(* IEC 61131-3 sources: SmartHomeNew/snapshots/2026-05-12 (part 2) *)

(* ---- FB_Time_Service.st ---- *)
FUNCTION_BLOCK FB_Time_Service
VAR
    L_Real_Now : UDINT;
    L_Elapsed : UDINT;
    L_Scaled_Delta : UDINT;
END_VAR

// read real time
L_Real_Now := GVL_STATUS.G_System_Time_MS;

// wrap-safe delta (real time base)
IF L_Real_Now >= GVL_TIME_SERVICE.G_Last_Now_MS THEN
    L_Elapsed := L_Real_Now - GVL_TIME_SERVICE.G_Last_Now_MS;
    GVL_TIME_SERVICE.G_Wrap_Detected := FALSE;
ELSE
    L_Elapsed := (16#FFFFFFFF - GVL_TIME_SERVICE.G_Last_Now_MS) + L_Real_Now + 1;
    GVL_TIME_SERVICE.G_Wrap_Detected := TRUE;
END_IF;

GVL_TIME_SERVICE.G_Last_Now_MS := L_Real_Now;

// --- SIMULATION MODE ---
IF GVL_TIME_SERVICE.G_Sim_Enabled THEN

    IF NOT GVL_TIME_SERVICE.G_Sim_Frozen THEN
        L_Scaled_Delta := REAL_TO_UDINT(TO_REAL(L_Elapsed) * GVL_TIME_SERVICE.G_Sim_Time_Scale);

        GVL_TIME_SERVICE.G_Sim_Now_MS := GVL_TIME_SERVICE.G_Sim_Now_MS + L_Scaled_Delta;

        GVL_TIME_SERVICE.G_Sim_Time_Of_Day_MS := GVL_TIME_SERVICE.G_Sim_Time_Of_Day_MS + L_Scaled_Delta;

        IF GVL_TIME_SERVICE.G_Sim_Time_Of_Day_MS >= 86400000 THEN
            GVL_TIME_SERVICE.G_Sim_Time_Of_Day_MS := GVL_TIME_SERVICE.G_Sim_Time_Of_Day_MS MOD 86400000;
            GVL_TIME_SERVICE.G_Sim_Day_Of_Week := GVL_TIME_SERVICE.G_Sim_Day_Of_Week + 1;
            IF GVL_TIME_SERVICE.G_Sim_Day_Of_Week > 7 THEN
                GVL_TIME_SERVICE.G_Sim_Day_Of_Week := 1;
            END_IF;
        END_IF;
    END_IF;

    GVL_TIME_SERVICE.G_Now_MS := GVL_TIME_SERVICE.G_Sim_Now_MS;
    GVL_TIME_SERVICE.G_Time_Of_Day_MS := GVL_TIME_SERVICE.G_Sim_Time_Of_Day_MS;
    GVL_TIME_SERVICE.G_Day_Of_Week := GVL_TIME_SERVICE.G_Sim_Day_Of_Week;

ELSE
    GVL_TIME_SERVICE.G_Now_MS := L_Real_Now;
    GVL_TIME_SERVICE.G_Time_Of_Day_MS := GVL_STATUS.G_Time_Of_Day_MS;
    GVL_TIME_SERVICE.G_Day_Of_Week := TO_INT(GVL_STATUS.G_Current_Day);
END_IF;

// TOD unified
GVL_TIME_SERVICE.G_Current_TOD := UDINT_TO_TOD(GVL_TIME_SERVICE.G_Time_Of_Day_MS);

GVL_TIME_SERVICE.G_Delta_MS := L_Elapsed;

END_FUNCTION_BLOCK

(* ---- FB_Water_Output_Projection.st ---- *)
FUNCTION_BLOCK FB_Water_Output_Projection
VAR_INPUT
    VI_Zone_Enable : ARRAY[1..32] OF BOOL;
    VI_Valve_35_Close : BOOL;
    VI_Valve_36_Close : BOOL;
END_VAR
VAR
    L_i : INT;
END_VAR

FOR L_i := 1 TO 32 DO
    GVL_WATER_OUTPUT.DO_Water_Zone_Enable[L_i] := VI_Zone_Enable[L_i];
END_FOR;

GVL_WATER_OUTPUT.DO_Water_Valve_35_Close := VI_Valve_35_Close;
GVL_WATER_OUTPUT.DO_Water_Valve_36_Close := VI_Valve_36_Close;

END_FUNCTION_BLOCK
// >>> BULK_SYNC_ANCHOR: FB_Water_Output_Projection <<<

(* ---- PRG_Command_Verifier.st ---- *)
PROGRAM PRG_Command_Verifier
VAR
    L_i : INT;
    L_Mismatch_Count : INT := 0;
    L_Runtime_Error : BOOL := FALSE;
    L_Runtime_Error_Code : UDINT := 0;
    L_Runtime_Error_Text : STRING(160) := '';
    L_Now_MS : UDINT;
    L_Prev_Runtime_Error : BOOL;
    L_Any_Manifold_Pump_On : BOOL;
    fbLog : FB_LogEvent;
END_VAR

L_Now_MS := GVL_STATUS.G_System_Time_MS;

// ===============================
// 1. COMMAND MISMATCH CHECK
// ===============================
L_Mismatch_Count := 0;

IF GVL_COMMAND.G_Gas_Valve_Close <> GVL_COMMAND_SHADOW.G_Gas_Valve_Close THEN L_Mismatch_Count := L_Mismatch_Count + 1; END_IF;
IF GVL_COMMAND.G_Boiler_Stop <> GVL_COMMAND_SHADOW.G_Boiler_Stop THEN L_Mismatch_Count := L_Mismatch_Count + 1; END_IF;
IF GVL_COMMAND.G_Vent_Stop <> GVL_COMMAND_SHADOW.G_Vent_Stop THEN L_Mismatch_Count := L_Mismatch_Count + 1; END_IF;
IF GVL_COMMAND.G_Supply_100_Req <> GVL_COMMAND_SHADOW.G_Supply_100_Req THEN L_Mismatch_Count := L_Mismatch_Count + 1; END_IF;
IF GVL_COMMAND.G_Supply_80_Req <> GVL_COMMAND_SHADOW.G_Supply_80_Req THEN L_Mismatch_Count := L_Mismatch_Count + 1; END_IF;
IF GVL_COMMAND.G_Vent_PV3_Boost <> GVL_COMMAND_SHADOW.G_Vent_PV3_Boost THEN L_Mismatch_Count := L_Mismatch_Count + 1; END_IF;
IF GVL_COMMAND.G_Close_Valve_35 <> GVL_COMMAND_SHADOW.G_Close_Valve_35 THEN L_Mismatch_Count := L_Mismatch_Count + 1; END_IF;
IF GVL_COMMAND.G_Close_Valve_36 <> GVL_COMMAND_SHADOW.G_Close_Valve_36 THEN L_Mismatch_Count := L_Mismatch_Count + 1; END_IF;
IF GVL_COMMAND.G_Lock_1_Open <> GVL_COMMAND_SHADOW.G_Lock_1_Open THEN L_Mismatch_Count := L_Mismatch_Count + 1; END_IF;
IF GVL_COMMAND.G_Lock_1_Close <> GVL_COMMAND_SHADOW.G_Lock_1_Close THEN L_Mismatch_Count := L_Mismatch_Count + 1; END_IF;
IF GVL_COMMAND.G_Lock_2_Open <> GVL_COMMAND_SHADOW.G_Lock_2_Open THEN L_Mismatch_Count := L_Mismatch_Count + 1; END_IF;
IF GVL_COMMAND.G_Lock_2_Close <> GVL_COMMAND_SHADOW.G_Lock_2_Close THEN L_Mismatch_Count := L_Mismatch_Count + 1; END_IF;
IF GVL_COMMAND.G_Gate_Open <> GVL_COMMAND_SHADOW.G_Gate_Open THEN L_Mismatch_Count := L_Mismatch_Count + 1; END_IF;
IF GVL_COMMAND.G_Wicket_Open <> GVL_COMMAND_SHADOW.G_Wicket_Open THEN L_Mismatch_Count := L_Mismatch_Count + 1; END_IF;

GVL_COMMAND_VERIFY.Command_Mismatch_Count := L_Mismatch_Count;
GVL_COMMAND_VERIFY.Command_Match_OK := (L_Mismatch_Count = 0);
GVL_COMMAND_VERIFY.Command_Mismatch_Active := (L_Mismatch_Count > 0);

// ===============================
// 2. RUNTIME SANITY CHECKS
// ===============================
L_Runtime_Error := FALSE;
L_Runtime_Error_Code := 0;
L_Runtime_Error_Text := '';
L_Any_Manifold_Pump_On := FALSE;

// PLC inactive: fail-safe outputs should be off/safe except alarm/gas close outputs.
IF (NOT L_Runtime_Error) AND (NOT GVL_STATUS.G_Is_Active_PLC) THEN
    FOR L_i := 1 TO GVL_CONSTANTS.C_MAX_HEATING_CIRCUITS DO
        IF GVL_IO.DO_Zone_Valves[L_i] THEN
            L_Runtime_Error := TRUE;
            L_Runtime_Error_Code := 10;
            L_Runtime_Error_Text := 'PLC inactive zone valve on';
        END_IF;
    END_FOR;
END_IF;

IF (NOT L_Runtime_Error) AND (NOT GVL_STATUS.G_Is_Active_PLC) THEN
    FOR L_i := 1 TO GVL_CONSTANTS.C_MAX_MANIFOLDS DO
        IF GVL_IO.DO_Manifold_Pumps[L_i] THEN
            L_Runtime_Error := TRUE;
            L_Runtime_Error_Code := 11;
            L_Runtime_Error_Text := 'PLC inactive pump on';
        END_IF;
    END_FOR;
END_IF;

// GAS: gas valve must be physically commanded closed.
IF (NOT L_Runtime_Error) AND (GVL_SAFETY_SHUTDOWN.G_Safety_Mode = GAS) AND (NOT GVL_IO.DO_Gas_Valve_Close) THEN
    L_Runtime_Error := TRUE;
    L_Runtime_Error_Code := 1;
    L_Runtime_Error_Text := 'Gas valve not closed';
END_IF;

// GAS: ventilation must not be forced fully off by the IO layer.
IF (NOT L_Runtime_Error) AND (GVL_SAFETY_SHUTDOWN.G_Safety_Mode = GAS) THEN
    IF (GVL_IO.AO_Supply_Fans[1] = 0) AND (GVL_IO.AO_Exhaust_Fans[1] = 0) THEN
        L_Runtime_Error := TRUE;
        L_Runtime_Error_Code := 3;
        L_Runtime_Error_Text := 'Gas ventilation inactive';
    END_IF;
END_IF;

// FIRE: all exhaust fans should be commanded above zero in smoke exhaust mode.
IF (NOT L_Runtime_Error) AND (GVL_SAFETY_SHUTDOWN.G_Safety_Mode = FIRE) THEN
    FOR L_i := 1 TO GVL_CONSTANTS.C_MAX_EXHAUST_FANS DO
        IF GVL_IO.AO_Exhaust_Fans[L_i] = 0 THEN
            L_Runtime_Error := TRUE;
            L_Runtime_Error_Code := 2;
            L_Runtime_Error_Text := 'Smoke exhaust not active';
        END_IF;
    END_FOR;
END_IF;

// FIRE: supply fans should be off in smoke exhaust mode.
IF (NOT L_Runtime_Error) AND (GVL_SAFETY_SHUTDOWN.G_Safety_Mode = FIRE) THEN
    FOR L_i := 1 TO GVL_CONSTANTS.C_MAX_SUPPLY_FANS DO
        IF GVL_IO.AO_Supply_Fans[L_i] <> 0 THEN
            L_Runtime_Error := TRUE;
            L_Runtime_Error_Code := 4;
            L_Runtime_Error_Text := 'Supply fan active in fire';
        END_IF;
    END_FOR;
END_IF;

// WATER_LEAK: valve close commands must reach physical outputs.
IF (NOT L_Runtime_Error) AND (GVL_SAFETY_SHUTDOWN.G_Safety_Mode = WATER_LEAK) THEN
    IF GVL_COMMAND_SHADOW.G_Close_Valve_35 AND (NOT GVL_IO.DO_Water_Valve_35_Close) THEN
        L_Runtime_Error := TRUE;
        L_Runtime_Error_Code := 5;
        L_Runtime_Error_Text := 'Water valve 35 not closed';
    ELSIF GVL_COMMAND_SHADOW.G_Close_Valve_36 AND (NOT GVL_IO.DO_Water_Valve_36_Close) THEN
        L_Runtime_Error := TRUE;
        L_Runtime_Error_Code := 6;
        L_Runtime_Error_Text := 'Water valve 36 not closed';
    END_IF;
END_IF;

// FREEZE: when freeze-risk is active, heating circulation should not be fully dead.
IF (NOT L_Runtime_Error) AND GVL_STATE.G_Safety_Freeze_Risk THEN
    FOR L_i := 1 TO GVL_CONSTANTS.C_MAX_MANIFOLDS DO
        IF GVL_IO.DO_Manifold_Pumps[L_i] THEN
            L_Any_Manifold_Pump_On := TRUE;
        END_IF;
    END_FOR;

    IF (NOT L_Any_Manifold_Pump_On) AND (NOT GVL_IO.DO_Backup_Circulation_Pump) THEN
        L_Runtime_Error := TRUE;
        L_Runtime_Error_Code := 7;
        L_Runtime_Error_Text := 'Freeze circulation inactive';
    END_IF;
END_IF;

// GAS+FREEZE: electric backup may be used for anti-freeze, but DHW heating must remain off.
IF (NOT L_Runtime_Error) AND GVL_STATE.G_Safety_Freeze_Risk AND GVL_COMMAND_SHADOW.G_Heating_Gas_Safety_Stop THEN
    IF GVL_IO.DO_DHW_Heating_Pump THEN
        L_Runtime_Error := TRUE;
        L_Runtime_Error_Code := 8;
        L_Runtime_Error_Text := 'DHW heating active during gas freeze';
    END_IF;
END_IF;

// Apply result
IF L_Runtime_Error THEN
    GVL_COMMAND_VERIFY.Runtime_Sanity_OK := FALSE;
    GVL_COMMAND_VERIFY.Runtime_Last_Error_Code := L_Runtime_Error_Code;
    GVL_COMMAND_VERIFY.Runtime_Last_Error_Text := L_Runtime_Error_Text;
    GVL_COMMAND_VERIFY.Runtime_Last_Error_Time_MS := L_Now_MS;
    GVL_CONFIG_VALIDATION.G_Runtime_Sanity_OK := FALSE;
    GVL_CONFIG_VALIDATION.G_Runtime_Sanity_Error := TRUE;
    GVL_CONFIG_VALIDATION.G_Runtime_Last_Error_Code := L_Runtime_Error_Code;
    GVL_CONFIG_VALIDATION.G_Runtime_Last_Error_Text := L_Runtime_Error_Text;
    GVL_CONFIG_VALIDATION.G_Runtime_Last_Error_MS := L_Now_MS;

    IF NOT L_Prev_Runtime_Error THEN
        GVL_COMMAND_VERIFY.Runtime_Sanity_Error_Count := GVL_COMMAND_VERIFY.Runtime_Sanity_Error_Count + 1;
        fbLog(
            VI_Event_Type := 1001,
            VI_Timestamp := L_Now_MS,
            VI_Param1 := L_Runtime_Error_Code,
            VI_Param2 := GVL_COMMAND_VERIFY.Runtime_Sanity_Error_Count
        );
    END_IF;
ELSE
    GVL_COMMAND_VERIFY.Runtime_Sanity_OK := TRUE;
    GVL_CONFIG_VALIDATION.G_Runtime_Sanity_OK := TRUE;
    GVL_CONFIG_VALIDATION.G_Runtime_Sanity_Error := FALSE;
END_IF;

L_Prev_Runtime_Error := L_Runtime_Error;

END_PROGRAM

(* ---- PRG_Config_Versioning.st ---- *)
PROGRAM PRG_Config_Versioning
VAR
    L_i : INT;
    L_Config_Error : BOOL;
END_VAR

// Detect config error from validation layer
L_Config_Error := GVL_STATUS.G_Diagnostics.Sensor_Fault OR GVL_STATUS.G_Diagnostics.Subsystem_Degraded;

// --- Save snapshot when system is healthy ---
IF NOT L_Config_Error THEN
    FOR L_i := 1 TO GVL_CONSTANTS.C_MAX_HEATING_CIRCUITS DO
        GVL_CONFIG_BACKUP.G_Backup_FloorHeating_Configs[L_i] := GVL_CONFIG.G_HMI_FloorHeating_Configs[L_i];
    END_FOR;

    GVL_CONFIG_BACKUP.G_Backup_Max_Active_Manifolds := GVL_CONFIG.G_Max_Active_Manifolds;
    GVL_CONFIG_BACKUP.G_Backup_Max_Thermal_Budget := GVL_CONFIG.G_Max_Thermal_Budget;

    GVL_CONFIG_BACKUP.G_Backup_Valid := TRUE;
END_IF;

// --- Rollback if config invalid ---
IF L_Config_Error THEN

    // Freeze system via command layer
    GVL_COMMAND_SHADOW.G_Heating_Block := TRUE;
    GVL_COMMAND_SHADOW.G_Boiler_Stop := TRUE;

    // Restore snapshot only if valid
    IF GVL_CONFIG_BACKUP.G_Backup_Valid THEN
        FOR L_i := 1 TO GVL_CONSTANTS.C_MAX_HEATING_CIRCUITS DO
            GVL_CONFIG.G_HMI_FloorHeating_Configs[L_i] := GVL_CONFIG_BACKUP.G_Backup_FloorHeating_Configs[L_i];
        END_FOR;

        GVL_CONFIG.G_Max_Active_Manifolds := GVL_CONFIG_BACKUP.G_Backup_Max_Active_Manifolds;
        GVL_CONFIG.G_Max_Thermal_Budget := GVL_CONFIG_BACKUP.G_Backup_Max_Thermal_Budget;

        GVL_STATUS.G_System_Mode_Text := 'CONFIG ROLLBACK';
    ELSE
        GVL_STATUS.G_System_Mode_Text := 'CONFIG INVALID - NO BACKUP';
    END_IF;
END_IF;

END_PROGRAM
// >>> BULK_SYNC_ANCHOR: PRG_Config_Versioning <<<

(* ---- PRG_Explainability.st ---- *)
PROGRAM PRG_Explainability
VAR
    L_Mode : E_Safety_Mode;
    L_Recovery : E_Recovery_Phase;
    L_Command : STRING(120);
    L_Heating : STRING(255);
END_VAR

L_Mode := GVL_SAFETY_SHUTDOWN.G_Safety_Mode;
L_Recovery := GVL_SAFETY_RECOVERY.G_Recovery_Phase;

GVL_EXPLAINABILITY.G_Last_Safety_Mode := L_Mode;
GVL_EXPLAINABILITY.G_Last_Recovery_Phase := L_Recovery;
GVL_EXPLAINABILITY.G_Last_Update_MS := GVL_TIME_SERVICE.G_Now_MS;

// SAFETY LEVEL
CASE L_Mode OF
    FIRE: GVL_EXPLAINABILITY.G_Reason_Chain_Safety := 'FIRE';
    GAS: GVL_EXPLAINABILITY.G_Reason_Chain_Safety := 'GAS';
    WATER_LEAK: GVL_EXPLAINABILITY.G_Reason_Chain_Safety := 'WATER';
    GLOBAL_STOP: GVL_EXPLAINABILITY.G_Reason_Chain_Safety := 'GLOBAL_STOP';
    ELSE
        IF GVL_SAFETY_RECOVERY.G_Recovery_Active THEN
            GVL_EXPLAINABILITY.G_Reason_Chain_Safety := 'RECOVERY';
        ELSE
            GVL_EXPLAINABILITY.G_Reason_Chain_Safety := 'NORMAL';
        END_IF;
END_CASE;

// BEHAVIOR LEVEL
GVL_EXPLAINABILITY.G_Reason_Chain_Behavior := GVL_INTENT_BEHAVIOR.I_Reason_Text;

// COMMAND LEVEL
IF GVL_COMMAND_SHADOW.G_Heating_Block THEN
    L_Command := 'Heating Blocked';
ELSIF GVL_COMMAND_SHADOW.G_Vent_Stop THEN
    L_Command := 'Vent Stopped';
ELSIF GVL_COMMAND_SHADOW.G_Water_Block THEN
    L_Command := 'Water Blocked';
ELSE
    L_Command := 'Command OK';
END_IF;
GVL_EXPLAINABILITY.G_Reason_Chain_Command := L_Command;

// HEATING DOMAIN EXPLAINABILITY
IF GVL_STATE.G_Heating_RootCause <> E_Heating_RootCause.RC_NONE THEN
    L_Heating := GVL_STATE.G_Heating_Confidence_Reason_Text;
ELSIF GVL_STATE.G_Heating_Cascade_Degraded THEN
    L_Heating := 'Heating cascade degraded';
ELSE
    L_Heating := 'Heating OK';
END_IF;
GVL_EXPLAINABILITY.G_Heating_Why_Blocked := L_Heating;

// OUTPUT LEVEL
GVL_EXPLAINABILITY.G_Reason_Chain_Output := 'Outputs Applied';

// FULL CHAIN
GVL_EXPLAINABILITY.G_Reason_Chain_Full := CONCAT(
    CONCAT(
        CONCAT(
            GVL_EXPLAINABILITY.G_Reason_Chain_Safety,
            ' -> '
        ),
        CONCAT(
            GVL_EXPLAINABILITY.G_Reason_Chain_Behavior,
            ' -> '
        )
    ),
    CONCAT(
        CONCAT(
            GVL_EXPLAINABILITY.G_Reason_Chain_Command,
            ' -> '
        ),
        CONCAT(
            L_Heating,
            ' -> Outputs Applied'
        )
    )
);

// KEEP OLD FIELDS
GVL_EXPLAINABILITY.G_Behavior_Why_Active := GVL_INTENT_BEHAVIOR.I_Reason_Text;

END_PROGRAM

(* ---- PRG_Heating.st ---- *)
PROGRAM PRG_Heating
VAR
    fbHeatingManager : FB_Heating_System_Manager;
    fbDHWManager : FB_DHW_Manager;
    fbOutputProjection : FB_Heating_Output_Projection;
    fbRootCauseDiagnostics : FB_Heating_RootCause_Diagnostics;
    fbHeatingDiagnostics : FB_Heating_Diagnostics;
    fbRuntimeObserver : FB_Heating_Runtime_Observer;
    fbRuntimeObserverAuthorization : FB_Heating_Runtime_Observer_Authorization;

    L_Runtime_Context : ST_Heating_Runtime_Context;

    L_Runtime_Observer_Enable_Last : BOOL := FALSE;
    L_Runtime_Observer_Activation_Stabilized : BOOL := FALSE;

    L_i : INT;
    L_Current_Hour : UINT;
    L_Boiler_Modulation_REAL : ARRAY[1..GVL_CONSTANTS.C_MAX_BOILERS] OF REAL;

    L_Heating_Emergency_Stop : BOOL;
    L_Heating_Gas_Safety_Stop : BOOL;

    L_Zone_Valves : ARRAY[1..GVL_CONSTANTS.C_MAX_HEATING_CIRCUITS] OF BOOL;
    L_Manifold_Pumps : ARRAY[1..GVL_CONSTANTS.C_MAX_MANIFOLDS] OF BOOL;
    L_Manifold_Valves : ARRAY[1..GVL_CONSTANTS.C_MAX_MANIFOLDS] OF REAL;
    L_Boiler_OT_Enable : ARRAY[1..GVL_CONSTANTS.C_MAX_BOILERS] OF BOOL;
    L_Boiler_OT_Setpoint : ARRAY[1..GVL_CONSTANTS.C_MAX_BOILERS] OF REAL;
    L_Backup_Circulation_Pump : BOOL;
    L_Electric_Heater_Enable : BOOL;
    L_Freeze_Risk_Status : BOOL;
    L_Manifold_Status : ARRAY[1..GVL_CONSTANTS.C_MAX_MANIFOLDS] OF ST_Manifold_Status;
    L_Boiler_Status : ARRAY[1..GVL_CONSTANTS.C_MAX_BOILERS] OF ST_Boiler_Status;
    L_DHW_Heating_Pump : BOOL;
    L_DHW_Circ_Pump : BOOL;
    L_DHW_Status : ST_DHW_Status;
END_VAR

FOR L_i := 1 TO GVL_CONSTANTS.C_MAX_BOILERS DO
    L_Boiler_Modulation_REAL[L_i] := TO_REAL(GVL_IO.AI_Boiler_Modulation[L_i]);
END_FOR;

L_Current_Hour := TO_UINT(GVL_TIME_SERVICE.G_Time_Of_Day_MS / 3600000);

L_Heating_Emergency_Stop := GVL_COMMAND_SHADOW.G_Heating_Emergency_Stop;
L_Heating_Gas_Safety_Stop := GVL_COMMAND_SHADOW.G_Heating_Gas_Safety_Stop OR GVL_STATE.G_Safety_Gas_Latched;

L_Runtime_Context.Runtime_Enabled := TRUE;
L_Runtime_Context.Runtime_Ready := TRUE;
L_Runtime_Context.Runtime_Fault := FALSE;
L_Runtime_Context.Current_Phase := E_Heating_Runtime_Phase.HRP_IDLE;

L_Runtime_Context.Allow_DHW_Phase := TRUE;
L_Runtime_Context.Allow_Heating_Phase := TRUE;
L_Runtime_Context.Allow_Service_Gating_Phase := TRUE;
L_Runtime_Context.Allow_State_Publication_Phase := TRUE;
L_Runtime_Context.Allow_Diagnostics_Phase := TRUE;
L_Runtime_Context.Allow_Output_Projection_Phase := TRUE;

L_Runtime_Context.DHW_Executed := FALSE;
L_Runtime_Context.Heating_Executed := FALSE;
L_Runtime_Context.Service_Gating_Executed := FALSE;
L_Runtime_Context.State_Publication_Executed := FALSE;
L_Runtime_Context.Diagnostics_Executed := FALSE;
L_Runtime_Context.Output_Projection_Executed := FALSE;

L_Runtime_Context.DHW_Before_Heating_Valid := TRUE;
L_Runtime_Context.State_Publication_Before_Diagnostics_Valid := TRUE;
L_Runtime_Context.Output_Projection_Last_Valid := TRUE;

L_Runtime_Context.Diagnostics_Isolation_Valid := TRUE;
L_Runtime_Context.Explainability_Isolation_Valid := TRUE;
L_Runtime_Context.Safety_Isolation_Valid := TRUE;
L_Runtime_Context.OpenTherm_Ownership_Valid := TRUE;
L_Runtime_Context.Cascade_Ownership_Valid := TRUE;

L_Runtime_Context.Runtime_Status_Code := 1;
L_Runtime_Context.Runtime_Status_Text := 'Heating runtime nominal';

// ======================================================
// GOVERNED OBSERVER AUTHORIZATION EVALUATION
// ======================================================
GVL_Heating_Runtime_Observer.G_Runtime_Observer_Lifecycle_State :=
    E_Runtime_Observer_Lifecycle_State.ROS_AUTHORIZATION_PENDING;
GVL_Heating_Runtime_Observation.G_Runtime_Observer_Lifecycle_State :=
    E_Runtime_Observer_Lifecycle_State.ROS_AUTHORIZATION_PENDING;
GVL_Heating_Runtime_Observation.G_Runtime_Observer_Lifecycle_Code := 10;
GVL_Heating_Runtime_Observation.G_Runtime_Observer_Lifecycle_Text :=
    'Heating runtime observer authorization pending';
GVL_Heating_Runtime_Observation.G_Runtime_Observer_Commissioning_Active :=
    GVL_Heating_Runtime_Observer.G_Runtime_Observer_Enable_Request;

fbRuntimeObserverAuthorization(
    VI_Enable_Request := GVL_Heating_Runtime_Observer.G_Runtime_Observer_Enable_Request,
    VI_Bootstrap_Mode := GVL_Heating_Runtime_Observer.G_Runtime_Observer_Bootstrap_Mode,
    VI_Passive_Mode := GVL_Heating_Runtime_Observer.G_Runtime_Observer_Passive_Mode,
    VI_ReadOnly_Mode := GVL_Heating_Runtime_Observer.G_Runtime_Observer_ReadOnly_Mode,
    VI_Governance_Locked := GVL_Heating_Runtime_Observer.G_Runtime_Observer_Governance_Locked,
    VI_Runtime_Authority_Disabled := GVL_Heating_Runtime_Observer.G_Runtime_Observer_Runtime_Authority_Disabled,
    VI_Writable_Exports_Disabled := GVL_Heating_Runtime_Observer.G_Runtime_Observer_Writable_Exports_Disabled
);

GVL_Heating_Runtime_Observer.G_Runtime_Observer_Enable_Authorized :=
    fbRuntimeObserverAuthorization.VO_Enable_Authorized;

GVL_Heating_Runtime_Observer.G_Runtime_Observer_Enable_Effective :=
    fbRuntimeObserverAuthorization.VO_Enable_Effective;

GVL_Heating_Runtime_Observer.G_Runtime_Observer_Authorization_Valid :=
    fbRuntimeObserverAuthorization.VO_Authorization_Valid;

GVL_Heating_Runtime_Observer.G_Runtime_Observer_Authorization_Status_Code :=
    fbRuntimeObserverAuthorization.VO_Status_Code;

GVL_Heating_Runtime_Observer.G_Runtime_Observer_Authorization_Status_Text :=
    fbRuntimeObserverAuthorization.VO_Status_Text;

IF NOT GVL_Heating_Runtime_Observer.G_Runtime_Observer_Enable_Request THEN
    GVL_Heating_Runtime_Observer.G_Runtime_Observer_Lifecycle_State :=
        E_Runtime_Observer_Lifecycle_State.ROS_INACTIVE;
    GVL_Heating_Runtime_Observation.G_Runtime_Observer_Lifecycle_State :=
        E_Runtime_Observer_Lifecycle_State.ROS_INACTIVE;
    GVL_Heating_Runtime_Observation.G_Runtime_Observer_Lifecycle_Code := 0;
    GVL_Heating_Runtime_Observation.G_Runtime_Observer_Lifecycle_Text :=
        'Heating runtime observer inactive';
    GVL_Heating_Runtime_Observation.G_Runtime_Observer_Commissioning_Active := FALSE;
ELSIF NOT GVL_Heating_Runtime_Observer.G_Runtime_Observer_Enable_Effective THEN
    GVL_Heating_Runtime_Observer.G_Runtime_Observer_Lifecycle_State :=
        E_Runtime_Observer_Lifecycle_State.ROS_AUTHORIZATION_DENIED;
    GVL_Heating_Runtime_Observation.G_Runtime_Observer_Lifecycle_State :=
        E_Runtime_Observer_Lifecycle_State.ROS_AUTHORIZATION_DENIED;
    GVL_Heating_Runtime_Observation.G_Runtime_Observer_Lifecycle_Code := 20;
    GVL_Heating_Runtime_Observation.G_Runtime_Observer_Lifecycle_Text :=
        'Heating runtime observer authorization denied';
END_IF;

L_Runtime_Context.Current_Phase := E_Heating_Runtime_Phase.HRP_DHW;

fbDHWManager(
    VI_System_Time_MS := GVL_STATUS.G_System_Time_MS,
    VI_Current_TOD := GVL_STATUS.G_Current_TOD,
    VI_IsActivePLC := GVL_STATUS.G_Is_Active_PLC,
    VI_Temp := GVL_STATE.G_DHW_Temp,
    VI_Pressure := GVL_STATE.G_DHW_Pressure,
    VI_Config := GVL_CONFIG.G_DHW_Config,
    VI_Current_Day_Of_Week := GVL_STATUS.G_Current_Day,
    VI_IO_Modules_Online := GVL_STATUS.G_IO_Modules_Online,
    VI_Reset_Errors := GVL_INTENT_USER.I_Reset_Errors,
    VI_Emergency_Stop := L_Heating_Emergency_Stop,
    VI_System_Mode := GVL_STATE.G_System_Mode,
    VO_Status => L_DHW_Status,
    VO_Heating_Pump => L_DHW_Heating_Pump,
    VO_Circ_Pump => L_DHW_Circ_Pump
);

L_Runtime_Context.DHW_Executed := TRUE;

IF L_Heating_Gas_Safety_Stop THEN
    L_DHW_Heating_Pump := FALSE;
    L_DHW_Status.Heating_Pump_On := FALSE;
END_IF;

L_Runtime_Context.Current_Phase := E_Heating_Runtime_Phase.HRP_HEATING;

fbHeatingManager(
    VI_System_Mode := GVL_STATE.G_System_Mode,
    VI_System_Time_MS := GVL_STATUS.G_System_Time_MS,
    VI_IsActivePLC := GVL_STATUS.G_Is_Active_PLC,
    VI_Outdoor_Temp := GVL_STATE.G_Outdoor_Temp,
    VI_Config := GVL_CONFIG.G_Heating_Config,
    VI_Tariff := GVL_CONFIG.G_HMI_Tariff_Settings,
    VI_Current_Hour := L_Current_Hour,
    VI_DHW_Heating_Demand := L_DHW_Heating_Pump,
    VI_DHW_Target_Temp := GVL_CONFIG.G_DHW_Config.Target_Temp,
    VI_Emergency_Stop := L_Heating_Emergency_Stop,
    VI_Gas_Safety_Stop := L_Heating_Gas_Safety_Stop,
    VI_Boiler_Error_Status := GVL_STATE.G_Boiler_Error,
    VI_Boiler_OT_Online := GVL_STATE.G_Boiler_OT_Online,
    VI_Boiler_Modulation := L_Boiler_Modulation_REAL,
    VI_Floor_Temps := GVL_STATE.G_Floor_Temps,
    VI_Room_Temps := GVL_STATE.G_Room_Temps,
    VI_Manifold_Pressures := GVL_STATE.G_Manifold_Pressures,
    VI_Manifold_Currents := GVL_STATE.G_Manifold_Currents,
    VI_Manifold_Temps_Supply := GVL_STATE.G_Manifold_T_Supply,
    VI_Manifold_Temps_Return := GVL_STATE.G_Manifold_T_Return,
    VI_Boiler_Flame_Status := GVL_STATE.G_Boiler_Flame,
    VI_Zone_Configs := GVL_CONFIG.G_HMI_FloorHeating_Configs,
    VI_Rule_Actions := GVL_STATE.G_Rule_Actions,
    VI_IO_Modules_Online := GVL_STATUS.G_IO_Modules_Online,
    VI_Manifold_End_Switches := GVL_STATE.G_Manifold_End_Switches,
    VI_Valve_Test_Config := GVL_CONFIG.G_Valve_Test_Config,
    VO_Manifold_Valves => L_Manifold_Valves,
    VO_Manifold_Pumps => L_Manifold_Pumps,
    VO_Zone_Valves => L_Zone_Valves,
    VO_Boiler_OT_Enable => L_Boiler_OT_Enable,
    VO_Boiler_OT_Setpoint => L_Boiler_OT_Setpoint,
    VO_Backup_Circulation_Pump => L_Backup_Circulation_Pump,
    VO_Electric_Heater_Enable => L_Electric_Heater_Enable,
    VO_Freeze_Risk_Status => L_Freeze_Risk_Status,
    VO_Status => L_Manifold_Status,
    VO_Boiler_Status => L_Boiler_Status
);

L_Runtime_Context.Heating_Executed := TRUE;

L_Runtime_Context.Current_Phase := E_Heating_Runtime_Phase.HRP_SERVICE_GATING;

GVL_STATUS.G_Diagnostics.Backup_Pump_Out_Of_Service := NOT GVL_CONFIG.G_Backup_Circulation_Pump_In_Service;
GVL_STATUS.G_Diagnostics.Electric_Heater_Out_Of_Service := NOT GVL_CONFIG.G_Electric_Heater_In_Service;

IF NOT GVL_CONFIG.G_Backup_Circulation_Pump_In_Service THEN
    L_Backup_Circulation_Pump := FALSE;
END_IF;

IF NOT GVL_CONFIG.G_Electric_Heater_In_Service THEN
    L_Electric_Heater_Enable := FALSE;
END_IF;

FOR L_i := 1 TO GVL_CONSTANTS.C_MAX_MANIFOLDS DO
    GVL_STATUS.G_Diagnostics.Manifold_Pump_Out_Of_Service[L_i] := NOT GVL_CONFIG.G_Manifold_Pump_In_Service[L_i];
    IF NOT GVL_CONFIG.G_Manifold_Pump_In_Service[L_i] THEN
        L_Manifold_Pumps[L_i] := FALSE;
    END_IF;
END_FOR;

GVL_STATUS.G_Diagnostics.DHW_Heating_Pump_Out_Of_Service := NOT GVL_CONFIG.G_DHW_Heating_Pump_In_Service;
IF NOT GVL_CONFIG.G_DHW_Heating_Pump_In_Service THEN
    L_DHW_Heating_Pump := FALSE;
    L_DHW_Status.Heating_Pump_On := FALSE;
END_IF;

GVL_STATUS.G_Diagnostics.DHW_Circ_Pump_Out_Of_Service := NOT GVL_CONFIG.G_DHW_Circ_Pump_In_Service;
IF NOT GVL_CONFIG.G_DHW_Circ_Pump_In_Service THEN
    L_DHW_Circ_Pump := FALSE;
    L_DHW_Status.Circ_Pump_On := FALSE;
END_IF;

GVL_STATE.G_Freeze_Hardware_Degraded := GVL_STATUS.G_Diagnostics.Backup_Pump_Fault OR GVL_STATUS.G_Diagnostics.Electric_Heater_Fault;
GVL_STATE.G_Freeze_Hardware_Failed := GVL_STATUS.G_Diagnostics.Backup_Pump_Fault AND GVL_STATUS.G_Diagnostics.Electric_Heater_Fault;

IF GVL_STATE.G_Freeze_Hardware_Failed THEN
    L_Backup_Circulation_Pump := FALSE;
    L_Electric_Heater_Enable := FALSE;
    L_Freeze_Risk_Status := TRUE;
END_IF;

L_Runtime_Context.Service_Gating_Executed := TRUE;

L_Runtime_Context.Current_Phase := E_Heating_Runtime_Phase.HRP_STATE_PUBLICATION;

FOR L_i := 1 TO GVL_CONSTANTS.C_MAX_HEATING_CIRCUITS DO
    GVL_STATE.G_Zone_Valves[L_i] := L_Zone_Valves[L_i];
END_FOR;

FOR L_i := 1 TO GVL_CONSTANTS.C_MAX_MANIFOLDS DO
    GVL_STATE.G_Manifold_Pumps[L_i] := L_Manifold_Pumps[L_i];
    GVL_STATE.G_Manifold_Valves[L_i] := L_Manifold_Valves[L_i];
    GVL_STATUS.G_Manifold_Status[L_i] := L_Manifold_Status[L_i];
END_FOR;

FOR L_i := 1 TO GVL_CONSTANTS.C_MAX_BOILERS DO
    GVL_STATE.G_Boiler_OT_Enable[L_i] := L_Boiler_OT_Enable[L_i];
    GVL_STATE.G_Boiler_OT_Setpoint[L_i] := L_Boiler_OT_Setpoint[L_i];
    GVL_STATUS.G_Boiler_Status[L_i] := L_Boiler_Status[L_i];
END_FOR;

GVL_STATE.G_Backup_Circulation_Pump := L_Backup_Circulation_Pump;
GVL_STATE.G_Electric_Heater_Enable := L_Electric_Heater_Enable;
GVL_STATE.G_Safety_Freeze_Risk := L_Freeze_Risk_Status;
GVL_STATE.G_DHW_Heating_Pump := L_DHW_Heating_Pump;
GVL_STATE.G_DHW_Circ_Pump := L_DHW_Circ_Pump;
GVL_STATUS.G_DHW_Status := L_DHW_Status;

L_Runtime_Context.State_Publication_Executed := TRUE;

L_Runtime_Context.Current_Phase := E_Heating_Runtime_Phase.HRP_DIAGNOSTICS;

fbRootCauseDiagnostics(
    VI_Enable := TRUE
);

fbHeatingDiagnostics(
    VI_System_Time_MS := GVL_STATUS.G_System_Time_MS
);

L_Runtime_Context.Diagnostics_Executed := TRUE;

// ======================================================
// GOVERNED FINALIZED-STATE RUNTIME OBSERVER
// ======================================================
IF GVL_Heating_Runtime_Observer.G_Runtime_Observer_Enable_Effective THEN

    GVL_Heating_Runtime_Observer.G_Runtime_Observer_Rollback_Validated := FALSE;

    IF NOT L_Runtime_Observer_Enable_Last THEN
        L_Runtime_Observer_Activation_Stabilized := FALSE;

        GVL_Heating_Runtime_Observer.G_Runtime_Observer_Lifecycle_State :=
            E_Runtime_Observer_Lifecycle_State.ROS_STABILIZATION;
        GVL_Heating_Runtime_Observation.G_Runtime_Observer_Lifecycle_State :=
            E_Runtime_Observer_Lifecycle_State.ROS_STABILIZATION;
        GVL_Heating_Runtime_Observation.G_Runtime_Observer_Lifecycle_Code := 30;
        GVL_Heating_Runtime_Observation.G_Runtime_Observer_Lifecycle_Text :=
            'Heating runtime observer stabilization active';

        GVL_Heating_Runtime_Observation.G_Runtime_Observer_Commissioning_Required := TRUE;
        GVL_Heating_Runtime_Observation.G_Runtime_Observer_Commissioning_Active := TRUE;
        GVL_Heating_Runtime_Observation.G_Runtime_Observer_Commissioning_Complete := FALSE;

        GVL_Heating_Runtime_Observation.G_Runtime_Observation_Publication_Valid := FALSE;
        GVL_Heating_Runtime_Observation.G_Runtime_Observation_Stabilization_Complete := FALSE;
        GVL_Heating_Runtime_Observation.G_Runtime_Observation_Operational := FALSE;

        GVL_Heating_Runtime_Observation.G_Runtime_Observation_Valid := FALSE;
        GVL_Heating_Runtime_Observation.G_Runtime_Observer_Ready := FALSE;
        GVL_Heating_Runtime_Observation.G_Runtime_Observer_Fault := FALSE;
        GVL_Heating_Runtime_Observation.G_Runtime_Observation_Status_Code := 100;
        GVL_Heating_Runtime_Observation.G_Runtime_Observation_Status_Text :=
            'Heating runtime observer stabilization cycle active';
    END_IF;

    fbRuntimeObserver(
        VI_Enable := TRUE,
        VI_Runtime_Context := L_Runtime_Context,
        VI_Diagnostics_Valid := TRUE
    );

    GVL_Heating_Runtime_Observation.G_Runtime_Observation :=
        fbRuntimeObserver.VO_Observation;

    IF L_Runtime_Observer_Activation_Stabilized THEN
        GVL_Heating_Runtime_Observer.G_Runtime_Observer_Lifecycle_State :=
            E_Runtime_Observer_Lifecycle_State.ROS_OPERATIONAL;
        GVL_Heating_Runtime_Observation.G_Runtime_Observer_Lifecycle_State :=
            E_Runtime_Observer_Lifecycle_State.ROS_OPERATIONAL;
        GVL_Heating_Runtime_Observation.G_Runtime_Observer_Lifecycle_Code := 40;
        GVL_Heating_Runtime_Observation.G_Runtime_Observer_Lifecycle_Text :=
            'Heating runtime observer operational';

        GVL_Heating_Runtime_Observation.G_Runtime_Observer_Commissioning_Required := FALSE;
        GVL_Heating_Runtime_Observation.G_Runtime_Observer_Commissioning_Active := FALSE;
        GVL_Heating_Runtime_Observation.G_Runtime_Observer_Commissioning_Complete := TRUE;

        GVL_Heating_Runtime_Observation.G_Runtime_Observation_Publication_Valid := TRUE;
        GVL_Heating_Runtime_Observation.G_Runtime_Observation_Stabilization_Complete := TRUE;
        GVL_Heating_Runtime_Observation.G_Runtime_Observation_Operational := TRUE;

        GVL_Heating_Runtime_Observation.G_Runtime_Observation_Valid := TRUE;
        GVL_Heating_Runtime_Observation.G_Runtime_Observer_Ready :=
            fbRuntimeObserver.VO_Observer_Ready;
        GVL_Heating_Runtime_Observation.G_Runtime_Observer_Fault :=
            fbRuntimeObserver.VO_Observer_Fault;
        GVL_Heating_Runtime_Observation.G_Runtime_Observation_Status_Code :=
            fbRuntimeObserver.VO_Status_Code;
        GVL_Heating_Runtime_Observation.G_Runtime_Observation_Status_Text :=
            fbRuntimeObserver.VO_Status_Text;

        GVL_Heating_Runtime_Observer.G_Runtime_Observer_Activation_Validated := TRUE;
        GVL_Heating_Runtime_Observer.G_Runtime_Observer_Sequencing_Validated := TRUE;
        GVL_Heating_Runtime_Observer.G_Runtime_Observer_Publication_Validated := TRUE;
    ELSE
        L_Runtime_Observer_Activation_Stabilized := TRUE;
    END_IF;

ELSE
    L_Runtime_Observer_Activation_Stabilized := FALSE;

    IF L_Runtime_Observer_Enable_Last THEN
        GVL_Heating_Runtime_Observer.G_Runtime_Observer_Lifecycle_State :=
            E_Runtime_Observer_Lifecycle_State.ROS_ROLLBACK;
        GVL_Heating_Runtime_Observation.G_Runtime_Observer_Lifecycle_State :=
            E_Runtime_Observer_Lifecycle_State.ROS_ROLLBACK;
        GVL_Heating_Runtime_Observation.G_Runtime_Observer_Lifecycle_Code := 50;
        GVL_Heating_Runtime_Observation.G_Runtime_Observer_Lifecycle_Text :=
            'Heating runtime observer rollback cleanup completed';
    ELSIF GVL_Heating_Runtime_Observer.G_Runtime_Observer_Enable_Request THEN
        GVL_Heating_Runtime_Observer.G_Runtime_Observer_Lifecycle_State :=
            E_Runtime_Observer_Lifecycle_State.ROS_AUTHORIZATION_DENIED;
        GVL_Heating_Runtime_Observation.G_Runtime_Observer_Lifecycle_State :=
            E_Runtime_Observer_Lifecycle_State.ROS_AUTHORIZATION_DENIED;
        GVL_Heating_Runtime_Observation.G_Runtime_Observer_Lifecycle_Code := 20;
        GVL_Heating_Runtime_Observation.G_Runtime_Observer_Lifecycle_Text :=
            'Heating runtime observer authorization denied';
    ELSE
        GVL_Heating_Runtime_Observer.G_Runtime_Observer_Lifecycle_State :=
            E_Runtime_Observer_Lifecycle_State.ROS_INACTIVE;
        GVL_Heating_Runtime_Observation.G_Runtime_Observer_Lifecycle_State :=
            E_Runtime_Observer_Lifecycle_State.ROS_INACTIVE;
        GVL_Heating_Runtime_Observation.G_Runtime_Observer_Lifecycle_Code := 0;
        GVL_Heating_Runtime_Observation.G_Runtime_Observer_Lifecycle_Text :=
            'Heating runtime observer inactive';
    END_IF;

    GVL_Heating_Runtime_Observation.G_Runtime_Observer_Commissioning_Required := TRUE;
    GVL_Heating_Runtime_Observation.G_Runtime_Observer_Commissioning_Active := FALSE;
    GVL_Heating_Runtime_Observation.G_Runtime_Observer_Commissioning_Complete := FALSE;

    GVL_Heating_Runtime_Observation.G_Runtime_Observation.Runtime_Active := FALSE;
    GVL_Heating_Runtime_Observation.G_Runtime_Observation.Runtime_Ready := FALSE;
    GVL_Heating_Runtime_Observation.G_Runtime_Observation.Runtime_Fault := FALSE;
    GVL_Heating_Runtime_Observation.G_Runtime_Observation.Current_Phase := E_Heating_Runtime_Phase.HRP_DISABLED;

    GVL_Heating_Runtime_Observation.G_Runtime_Observation.DHW_Demand_Active := FALSE;
    GVL_Heating_Runtime_Observation.G_Runtime_Observation.DHW_Heating_Active := FALSE;
    GVL_Heating_Runtime_Observation.G_Runtime_Observation.DHW_Circulation_Active := FALSE;

    GVL_Heating_Runtime_Observation.G_Runtime_Observation.Heating_Demand_Active := FALSE;
    GVL_Heating_Runtime_Observation.G_Runtime_Observation.Heating_Runtime_Active := FALSE;
    GVL_Heating_Runtime_Observation.G_Runtime_Observation.Heating_Output_Active := FALSE;

    GVL_Heating_Runtime_Observation.G_Runtime_Observation.Cascade_Available := FALSE;
    GVL_Heating_Runtime_Observation.G_Runtime_Observation.Cascade_Degraded := FALSE;
    GVL_Heating_Runtime_Observation.G_Runtime_Observation.Cascade_Active_Boilers := 0;
    GVL_Heating_Runtime_Observation.G_Runtime_Observation.Cascade_Available_Boilers := 0;

    GVL_Heating_Runtime_Observation.G_Runtime_Observation.OpenTherm_Online := FALSE;
    GVL_Heating_Runtime_Observation.G_Runtime_Observation.OpenTherm_Command_Valid := FALSE;
    GVL_Heating_Runtime_Observation.G_Runtime_Observation.OpenTherm_Transport_Degraded := FALSE;

    GVL_Heating_Runtime_Observation.G_Runtime_Observation.Diagnostics_Active := FALSE;
    GVL_Heating_Runtime_Observation.G_Runtime_Observation.Explainability_Active := FALSE;

    GVL_Heating_Runtime_Observation.G_Runtime_Observation.DHW_Before_Heating_Observed := FALSE;
    GVL_Heating_Runtime_Observation.G_Runtime_Observation.Diagnostics_After_Publication_Observed := FALSE;
    GVL_Heating_Runtime_Observation.G_Runtime_Observation.Output_Projection_Last_Observed := FALSE;

    GVL_Heating_Runtime_Observation.G_Runtime_Observation.Runtime_Ownership_Valid := FALSE;
    GVL_Heating_Runtime_Observation.G_Runtime_Observation.Diagnostics_Ownership_Valid := FALSE;
    GVL_Heating_Runtime_Observation.G_Runtime_Observation.OpenTherm_Ownership_Valid := FALSE;
    GVL_Heating_Runtime_Observation.G_Runtime_Observation.Cascade_Ownership_Valid := FALSE;
    GVL_Heating_Runtime_Observation.G_Runtime_Observation.Safety_Ownership_Valid := FALSE;

    GVL_Heating_Runtime_Observation.G_Runtime_Observation.Observation_Status_Code := 0;
    GVL_Heating_Runtime_Observation.G_Runtime_Observation.Observation_Status_Text :=
        'Heating runtime observation inactive';

    GVL_Heating_Runtime_Observation.G_Runtime_Observation_Publication_Valid := FALSE;
    GVL_Heating_Runtime_Observation.G_Runtime_Observation_Stabilization_Complete := FALSE;
    GVL_Heating_Runtime_Observation.G_Runtime_Observation_Operational := FALSE;

    GVL_Heating_Runtime_Observation.G_Runtime_Observation_Valid := FALSE;
    GVL_Heating_Runtime_Observation.G_Runtime_Observer_Ready := FALSE;
    GVL_Heating_Runtime_Observation.G_Runtime_Observer_Fault := FALSE;
    GVL_Heating_Runtime_Observation.G_Runtime_Observation_Status_Code := 0;
    GVL_Heating_Runtime_Observation.G_Runtime_Observation_Status_Text :=
        'Heating runtime observation inactive';

    GVL_Heating_Runtime_Observer.G_Runtime_Observer_Activation_Validated := FALSE;
    GVL_Heating_Runtime_Observer.G_Runtime_Observer_Sequencing_Validated := FALSE;
    GVL_Heating_Runtime_Observer.G_Runtime_Observer_Publication_Validated := FALSE;
    GVL_Heating_Runtime_Observer.G_Runtime_Observer_Rollback_Validated := TRUE;
END_IF;

L_Runtime_Observer_Enable_Last :=
    GVL_Heating_Runtime_Observer.G_Runtime_Observer_Enable_Effective;

L_Runtime_Context.Current_Phase := E_Heating_Runtime_Phase.HRP_OUTPUT_PROJECTION;

fbOutputProjection(
    VI_Zone_Valves := L_Zone_Valves,
    VI_Manifold_Pumps := L_Manifold_Pumps,
    VI_Manifold_Valves := L_Manifold_Valves,
    VI_DHW_Heating_Pump := L_DHW_Heating_Pump,
    VI_DHW_Circ_Pump := L_DHW_Circ_Pump,
    VI_Backup_Circulation_Pump := L_Backup_Circulation_Pump,
    VI_Electric_Heater_Enable := L_Electric_Heater_Enable
);

L_Runtime_Context.Output_Projection_Executed := TRUE;
L_Runtime_Context.Current_Phase := E_Heating_Runtime_Phase.HRP_COMPLETE;

// >>> BULK_SYNC_ANCHOR: PRG_Heating <<<
END_PROGRAM

(* ---- PRG_OpenTherm_Transport.st ---- *)
PROGRAM PRG_OpenTherm_Transport
VAR
    L_i : INT;
    L_Status_Word : WORD;
    L_Heartbeat : UDINT;
    L_Ack_Seq : UDINT;
END_VAR

// ======================================================
// REAL TRANSPORT LAYER CONTRACT
// ======================================================
// This layer converts high-level command/status structures
// into transport-safe wire images.
//
// Real Modbus RTU/TCP or serial IO code must:
//   1. Write G_Wire_Image command fields to adapter registers.
//   2. Read adapter status registers into G_Wire_Image status fields.
//
// This program keeps protocol encoding/decoding centralized.
// It does not claim transport online unless OpenTherm is enabled.
// ======================================================

IF NOT GVL_CONFIG.G_OpenTherm_Enabled THEN
    GVL_OPENTHERM_ADAPTER.G_Transport_Online := FALSE;
    GVL_OPENTHERM_ADAPTER.G_Transport_Error := FALSE;

    FOR L_i := 1 TO GVL_CONSTANTS.C_MAX_BOILERS DO
        GVL_OPENTHERM_ADAPTER.G_Wire_Image[L_i].Cmd_Enable := 0;
        GVL_OPENTHERM_ADAPTER.G_Wire_Image[L_i].Cmd_Setpoint_x10 := 0;
        GVL_OPENTHERM_ADAPTER.G_Wire_Image[L_i].Cmd_Seq_Lo := 0;
        GVL_OPENTHERM_ADAPTER.G_Wire_Image[L_i].Cmd_Seq_Hi := 0;

        GVL_OPENTHERM_ADAPTER.G_Status[L_i].Raw_Online := FALSE;
        GVL_OPENTHERM_ADAPTER.G_Status[L_i].Raw_Error := FALSE;
        GVL_OPENTHERM_ADAPTER.G_Status[L_i].Raw_Flame := FALSE;
        GVL_OPENTHERM_ADAPTER.G_Status[L_i].Raw_Status_Word := 0;
    END_FOR;

    RETURN;
END_IF;

GVL_OPENTHERM_ADAPTER.G_Transport_Online := TRUE;
GVL_OPENTHERM_ADAPTER.G_Transport_Error := FALSE;
GVL_OPENTHERM_ADAPTER.G_Last_Transport_Update_MS := GVL_STATUS.G_System_Time_MS;

FOR L_i := 1 TO GVL_CONSTANTS.C_MAX_BOILERS DO

    // ======================================================
    // COMMAND → WIRE IMAGE
    // ======================================================
    IF GVL_OPENTHERM_ADAPTER.G_Command[L_i].Enable THEN
        GVL_OPENTHERM_ADAPTER.G_Wire_Image[L_i].Cmd_Enable := 1;
    ELSE
        GVL_OPENTHERM_ADAPTER.G_Wire_Image[L_i].Cmd_Enable := 0;
    END_IF;

    GVL_OPENTHERM_ADAPTER.G_Wire_Image[L_i].Cmd_Setpoint_x10 :=
        GVL_OPENTHERM_ADAPTER.G_Command[L_i].Setpoint_x10;

    GVL_OPENTHERM_ADAPTER.G_Wire_Image[L_i].Cmd_Seq_Lo :=
        UDINT_TO_WORD(GVL_OPENTHERM_ADAPTER.G_Command[L_i].Sequence AND 16#FFFF);

    GVL_OPENTHERM_ADAPTER.G_Wire_Image[L_i].Cmd_Seq_Hi :=
        UDINT_TO_WORD(SHR(GVL_OPENTHERM_ADAPTER.G_Command[L_i].Sequence, 16));

    // ======================================================
    // WIRE IMAGE → STATUS
    // ======================================================
    L_Heartbeat :=
        WORD_TO_UDINT(GVL_OPENTHERM_ADAPTER.G_Wire_Image[L_i].Status_Heartbeat_Lo)
        OR SHL(
            WORD_TO_UDINT(GVL_OPENTHERM_ADAPTER.G_Wire_Image[L_i].Status_Heartbeat_Hi),
            16
        );

    L_Ack_Seq :=
        WORD_TO_UDINT(GVL_OPENTHERM_ADAPTER.G_Wire_Image[L_i].Status_Ack_Seq_Lo)
        OR SHL(
            WORD_TO_UDINT(GVL_OPENTHERM_ADAPTER.G_Wire_Image[L_i].Status_Ack_Seq_Hi),
            16
        );

    GVL_OPENTHERM_ADAPTER.G_Status[L_i].Raw_Heartbeat := L_Heartbeat;
    GVL_OPENTHERM_ADAPTER.G_Status[L_i].Raw_Ack_Seq := L_Ack_Seq;

    L_Status_Word :=
        GVL_OPENTHERM_ADAPTER.G_Wire_Image[L_i].Status_Word;

    GVL_OPENTHERM_ADAPTER.G_Status[L_i].Raw_Online :=
        (L_Status_Word AND 16#0001) <> 0;

    GVL_OPENTHERM_ADAPTER.G_Status[L_i].Raw_Error :=
        (L_Status_Word AND 16#0002) <> 0;

    GVL_OPENTHERM_ADAPTER.G_Status[L_i].Raw_Flame :=
        (L_Status_Word AND 16#0004) <> 0;

    GVL_OPENTHERM_ADAPTER.G_Status[L_i].Raw_Status_Word :=
        L_Status_Word;

    GVL_OPENTHERM_ADAPTER.G_Status[L_i].Raw_Error_Code :=
        GVL_OPENTHERM_ADAPTER.G_Wire_Image[L_i].Error_Code;

    GVL_OPENTHERM_ADAPTER.G_Status[L_i].Raw_Modulation_x10 :=
        GVL_OPENTHERM_ADAPTER.G_Wire_Image[L_i].Modulation_x10;

    GVL_OPENTHERM_ADAPTER.G_Status[L_i].Raw_Boiler_Temp_x10 :=
        WORD_TO_INT(GVL_OPENTHERM_ADAPTER.G_Wire_Image[L_i].Boiler_Temp_x10);

END_FOR;

END_PROGRAM

(* ---- PRG_Security.st ---- *)
PROGRAM PRG_Security
VAR
    L_i : INT;
    L_Motion_Sensors_16 : ARRAY[1..16] OF BOOL;
    fbSecurityManager : FB_Security_System_Manager;
    fbAccessControl : FB_Access_Control;
END_VAR

FOR L_i := 1 TO 16 DO
    L_Motion_Sensors_16[L_i] := GVL_STATE.G_Motion_Sensors[L_i];
END_FOR;
// 7. Система безопасности (Охранная сигнализация)
fbSecurityManager(
    VI_System_Time_MS := GVL_STATUS.G_System_Time_MS,
    VI_IsActivePLC := GVL_STATUS.G_Is_Active_PLC,
    VI_Motion_Sensors := L_Motion_Sensors_16,
    VI_Door_Sensors := GVL_STATE.G_Door_Sensors,
    VI_Window_Sensors := GVL_STATE.G_Window_Sensors,
    VI_Arm_Request := GVL_INTENT_USER.I_Arm_Request,
    VI_Disarm_Request := GVL_INTENT_USER.I_Disarm_Request,
    VI_PIN_Code := GVL_INTENT_USER.I_PIN_Code,
    VI_RFID_Tag := GVL_INTENT_USER.I_RFID_Tag,
    VI_2FA_Code := GVL_INTENT_USER.I_2FA_Code_In,
    VI_Config := GVL_CONFIG.G_Security_Config,
    VI_Bypass_Motion := GVL_CONFIG.G_Security_Config.bypass_motion,
    VI_Bypass_Doors := GVL_CONFIG.G_Security_Config.bypass_doors,
    VI_Bypass_Windows := GVL_CONFIG.G_Security_Config.bypass_windows,
    VI_Current_TOD := GVL_STATUS.G_Current_TOD,
    VO_Armed => GVL_ALARM.G_Security_Armed,
    VO_Alarm_Active => GVL_ALARM.G_Security_Alarm,
    VO_Siren_Active => GVL_ALARM.G_Security_Siren,
    VO_Status_Msg => GVL_STATUS.G_Security_Status_Msg,
    VO_Send_Code_Req => GVL_COMMAND.G_Send_2FA_Req,
    VO_Code_To_Send => GVL_COMMAND.G_2FA_Code_Out
);

// 7.1 Контроль доступа (СКУД)
fbAccessControl(
    VI_System_Time_MS := GVL_STATUS.G_System_Time_MS,
    VI_IsActivePLC := GVL_STATUS.G_Is_Active_PLC,
    VI_Armed := GVL_ALARM.G_Security_Armed,
    VI_System_Mode := GVL_STATE.G_System_Mode,
    VI_Gate_Open_Req := GVL_CONFIG.G_HMI_Gate_Open_Req,
    VI_Wicket_Open_Req := GVL_CONFIG.G_HMI_Wicket_Open_Req,
    VI_Lock_1_Open_Req := GVL_CONFIG.G_HMI_Lock_1_Open_Req,
    VI_Lock_1_Close_Req := GVL_CONFIG.G_HMI_Lock_1_Close_Req,
    VI_Lock_2_Open_Req := GVL_CONFIG.G_HMI_Lock_2_Open_Req,
    VI_Lock_2_Close_Req := GVL_CONFIG.G_HMI_Lock_2_Close_Req,
    VI_PIN_Code := GVL_INTENT_USER.I_PIN_Code,
    VI_RFID_Tag := GVL_INTENT_USER.I_RFID_Tag,
    VI_Access_Codes := GVL_Retain.G_Access_Codes,
    VI_RFID_Tags := GVL_Retain.G_RFID_Tags,
    VI_Config := GVL_CONFIG.G_Security_Config,
    VO_Gate_Open => GVL_INTENT_USER.I_Gate_Open_Request,
    VO_Wicket_Open => GVL_INTENT_USER.I_Wicket_Open_Request,
    VO_Lock_1_Open => GVL_INTENT_USER.I_Lock_1_Open_Request,
    VO_Lock_1_Close => GVL_INTENT_USER.I_Lock_1_Close_Request,
    VO_Lock_2_Open => GVL_INTENT_USER.I_Lock_2_Open_Request,
    VO_Lock_2_Close => GVL_INTENT_USER.I_Lock_2_Close_Request
);
END_PROGRAM

(* ---- PRG_System_Diagnostics_Ext.st ---- *)
PROGRAM PRG_System_Diagnostics_Ext
VAR
    L_Error_Heating : BOOL;
    L_Error_Safety : BOOL;
    L_Error_IO : BOOL;

    L_Delta_Time : REAL;
    L_Now : UDINT;
    L_Last : UDINT;

    // cycle stats
    L_Cycle_MS : UDINT;
    L_Prev_Overrun : BOOL;
    L_Prev_Critical : BOOL;
    fbLog : FB_LogEvent;
END_VAR

L_Now := GVL_TIME_SERVICE.G_Now_MS;
L_Last := GVL_DIAGNOSTICS_EXT.G_Last_Update_Time;

// ===============================
// CYCLE INTERVAL MEASUREMENT
// ===============================
IF L_Last = 0 THEN
    L_Cycle_MS := GVL_DIAGNOSTICS_EXT.G_Cycle_Expected_MS;
ELSE
    IF L_Now >= L_Last THEN
        L_Cycle_MS := L_Now - L_Last;
    ELSE
        L_Cycle_MS := (4294967295 - L_Last) + L_Now + 1;
    END_IF;
END_IF;

GVL_DIAGNOSTICS_EXT.G_Last_Update_Time := L_Now;
GVL_DIAGNOSTICS_EXT.G_Cycle_Last_MS := L_Cycle_MS;

// min/max
IF (GVL_DIAGNOSTICS_EXT.G_Cycle_Min_MS = 0) OR (L_Cycle_MS < GVL_DIAGNOSTICS_EXT.G_Cycle_Min_MS) THEN
    GVL_DIAGNOSTICS_EXT.G_Cycle_Min_MS := L_Cycle_MS;
END_IF;

IF L_Cycle_MS > GVL_DIAGNOSTICS_EXT.G_Cycle_Max_MS THEN
    GVL_DIAGNOSTICS_EXT.G_Cycle_Max_MS := L_Cycle_MS;
END_IF;

// average (incremental)
GVL_DIAGNOSTICS_EXT.G_Cycle_Sample_Count := GVL_DIAGNOSTICS_EXT.G_Cycle_Sample_Count + 1;
GVL_DIAGNOSTICS_EXT.G_Cycle_Avg_MS :=
    GVL_DIAGNOSTICS_EXT.G_Cycle_Avg_MS +
    (UDINT_TO_REAL(L_Cycle_MS) - GVL_DIAGNOSTICS_EXT.G_Cycle_Avg_MS) /
    UDINT_TO_REAL(GVL_DIAGNOSTICS_EXT.G_Cycle_Sample_Count);

// ===============================
// OVERRUN / CRITICAL DETECTION
// ===============================
GVL_DIAGNOSTICS_EXT.G_Cycle_Overrun_Active := (L_Cycle_MS > GVL_DIAGNOSTICS_EXT.G_Cycle_Warning_MS);
GVL_DIAGNOSTICS_EXT.G_Cycle_Critical_Active := (L_Cycle_MS > GVL_DIAGNOSTICS_EXT.G_Cycle_Critical_MS);

IF GVL_DIAGNOSTICS_EXT.G_Cycle_Overrun_Active THEN
    GVL_DIAGNOSTICS_EXT.G_Cycle_Overrun_Count := GVL_DIAGNOSTICS_EXT.G_Cycle_Overrun_Count + 1;
    GVL_DIAGNOSTICS_EXT.G_Cycle_Last_Overrun_MS := L_Cycle_MS;
    GVL_DIAGNOSTICS_EXT.G_Cycle_Last_Overrun_Time_MS := L_Now;
END_IF;

IF GVL_DIAGNOSTICS_EXT.G_Cycle_Critical_Active THEN
    GVL_DIAGNOSTICS_EXT.G_Cycle_Critical_Count := GVL_DIAGNOSTICS_EXT.G_Cycle_Critical_Count + 1;
END_IF;

// edge logging
IF GVL_DIAGNOSTICS_EXT.G_Cycle_Overrun_Active AND NOT L_Prev_Overrun THEN
    fbLog(
        VI_Event_Type := 2001,
        VI_Timestamp := L_Now,
        VI_Param1 := L_Cycle_MS,
        VI_Param2 := GVL_DIAGNOSTICS_EXT.G_Cycle_Overrun_Count
    );
END_IF;

IF GVL_DIAGNOSTICS_EXT.G_Cycle_Critical_Active AND NOT L_Prev_Critical THEN
    fbLog(
        VI_Event_Type := 2002,
        VI_Timestamp := L_Now,
        VI_Param1 := L_Cycle_MS,
        VI_Param2 := GVL_DIAGNOSTICS_EXT.G_Cycle_Critical_Count
    );
END_IF;

L_Prev_Overrun := GVL_DIAGNOSTICS_EXT.G_Cycle_Overrun_Active;
L_Prev_Critical := GVL_DIAGNOSTICS_EXT.G_Cycle_Critical_Active;

// ===============================
// EXISTING HEALTH LOGIC
// ===============================
IF L_Last = 0 THEN
    L_Delta_Time := 0.1;
ELSE
    L_Delta_Time := UDINT_TO_REAL(L_Cycle_MS) / 1000.0;
END_IF;

L_Error_Heating := GVL_STATE.G_Heating_Subsystem_Degraded;
L_Error_Safety := GVL_STATE.G_Safety_Gas_Alarm OR GVL_STATE.G_Safety_Leak_Alarm OR GVL_STATE.G_Safety_Smoke_Alarm;
L_Error_IO := GVL_STATE.G_Heating_IO_Fault;

IF L_Error_Heating THEN
    GVL_DIAGNOSTICS_EXT.G_Error_Count_Heating := GVL_DIAGNOSTICS_EXT.G_Error_Count_Heating + 1;
    GVL_DIAGNOSTICS_EXT.G_Last_Error_Time_Heating := L_Now;
    GVL_DIAGNOSTICS_EXT.G_Health_Heating := GVL_DIAGNOSTICS_EXT.G_Health_Heating - (0.5 * L_Delta_Time);
ELSE
    GVL_DIAGNOSTICS_EXT.G_Health_Heating := GVL_DIAGNOSTICS_EXT.G_Health_Heating + (0.1 * L_Delta_Time);
END_IF;

IF L_Error_Safety THEN
    GVL_DIAGNOSTICS_EXT.G_Error_Count_Safety := GVL_DIAGNOSTICS_EXT.G_Error_Count_Safety + 1;
    GVL_DIAGNOSTICS_EXT.G_Last_Error_Time_Safety := L_Now;
    GVL_DIAGNOSTICS_EXT.G_Health_Safety := GVL_DIAGNOSTICS_EXT.G_Health_Safety - (1.0 * L_Delta_Time);
ELSE
    GVL_DIAGNOSTICS_EXT.G_Health_Safety := GVL_DIAGNOSTICS_EXT.G_Health_Safety + (0.2 * L_Delta_Time);
END_IF;

IF L_Error_IO THEN
    GVL_DIAGNOSTICS_EXT.G_Error_Count_IO := GVL_DIAGNOSTICS_EXT.G_Error_Count_IO + 1;
    GVL_DIAGNOSTICS_EXT.G_Last_Error_Time_IO := L_Now;
    GVL_DIAGNOSTICS_EXT.G_Health_IO := GVL_DIAGNOSTICS_EXT.G_Health_IO - (0.5 * L_Delta_Time);
ELSE
    GVL_DIAGNOSTICS_EXT.G_Health_IO := GVL_DIAGNOSTICS_EXT.G_Health_IO + (0.1 * L_Delta_Time);
END_IF;

// clamp
IF GVL_DIAGNOSTICS_EXT.G_Health_Heating < 0.0 THEN GVL_DIAGNOSTICS_EXT.G_Health_Heating := 0.0; END_IF;
IF GVL_DIAGNOSTICS_EXT.G_Health_Heating > 1.0 THEN GVL_DIAGNOSTICS_EXT.G_Health_Heating := 1.0; END_IF;

IF GVL_DIAGNOSTICS_EXT.G_Health_Safety < 0.0 THEN GVL_DIAGNOSTICS_EXT.G_Health_Safety := 0.0; END_IF;
IF GVL_DIAGNOSTICS_EXT.G_Health_Safety > 1.0 THEN GVL_DIAGNOSTICS_EXT.G_Health_Safety := 1.0; END_IF;

IF GVL_DIAGNOSTICS_EXT.G_Health_IO < 0.0 THEN GVL_DIAGNOSTICS_EXT.G_Health_IO := 0.0; END_IF;
IF GVL_DIAGNOSTICS_EXT.G_Health_IO > 1.0 THEN GVL_DIAGNOSTICS_EXT.G_Health_IO := 1.0; END_IF;

END_PROGRAM
